FUNCTION_BLOCK FB_MotionAxisResetNC IMPLEMENTS I_MotionAxisReset
VAR
    fbReset : MC_Reset;
END_VAR

END_FUNCTION_BLOCK

(* stored: Version 1.1.0.1
   POU FB_MotionAxisResetNC: Id {47868a8d-efc1-4ec3-95c0-016a2609019c}, SpecialFunc None *)
